// TwinCAT 3 PLC project PlcIotHttpSamplesPhilipsHue
// ProgramVersion: 3.1.4026.25
// libraries:
//   Tc2_Standard, * (Beckhoff Automation GmbH)
//   Tc2_System, * (Beckhoff Automation GmbH)
//   Tc2_Utilities, * (Beckhoff Automation GmbH)
//   Tc3_IotBase, * (Beckhoff Automation GmbH)
//   Tc3_JsonXml, * (Beckhoff Automation GmbH)
//   Tc3_Module, * (Beckhoff Automation GmbH)
// project tree:
//   / PlcTask.TcTTO (not stored)
//   POUs/ MAIN.TcPOU
//   POUs/Philips Hue/ FB_TestHTTP_Put_PhilipsHue.TcPOU
// real-time tasks:
//   TASK PlcTask: cycle T#10ms, priority 24, ADS port 350

// ---- POUs/MAIN.TcPOU
PROGRAM MAIN
VAR
	// trigger command execution for Philips Hue samples
	bPutPhilipsHue 					: BOOL;

	fbHttpClientPhilipsHue			: FB_IotHttpClient := (sHostName := '192.168.0.100',
									bKeepAlive := TRUE, tConnectionTimeout := T#10S);

	fbHttpPutPhilipsHue				: FB_TestHTTP_Put_PhilipsHue;
	
	bBlinkingMode					: BOOL;
	fbTimer							: TON:=(PT:=T#500MS);
	nColor               			: UINT;
END_VAR

// init client parameters at startup
IF NOT fbHttpClientPhilipsHue.bConfigured THEN 
	fbHttpClientPhilipsHue.nHostPort := 443;
	fbHttpClientPhilipsHue.stTLS.bNoServerCertCheck := TRUE;
END_IF

IF fbHttpClientPhilipsHue.bConfigured THEN
	fbHttpPutPhilipsHue(bSend := bPutPhilipsHue, fbClient := fbHttpClientPhilipsHue, nColor := nColor);
END_IF

IF bBlinkingMode THEN
	fbTimer(IN := NOT fbTimer.Q);
	IF fbTimer.Q THEN
		nColor := nColor +5000;
		IF nColor = 65000 THEN
			nColor :=0;
		END_IF
		IF bPutPhilipsHue THEN
			bPutPhilipsHue := FALSE;
		ELSE 
			bPutPhilipsHue := TRUE;
		END_IF
	END_IF
END_IF

fbHttpClientPhilipsHue.Execute();

END_PROGRAM

// ---- POUs/Philips Hue/FB_TestHTTP_Put_PhilipsHue.TcPOU
FUNCTION_BLOCK FB_TestHTTP_Put_PhilipsHue
VAR_INPUT
	bSend				: BOOL;
	nColor				: UINT;
END_VAR
VAR_IN_OUT
	fbClient			: FB_IotHttpClient;
END_VAR
VAR_OUTPUT
	bBusy				: BOOL;
	bError				: BOOL;
END_VAR
VAR
	fbRequest			: FB_IotHttpRequest;
	fbJson				: FB_JsonDomParser;
	fbJsonWriter		: FB_JsonSaxWriter;
	nState				: UDINT;
	RisingEdge			: R_TRIG;
	
	bGetContentResult	: BOOL;
	sContent			: STRING(511);
	sSend				: STRING(255);
	
	bGetJsonResult		: BOOL;
	jsonDoc				: SJsonValue;
	
	nReqCount			: UDINT;	
	nResCount			: UDINT;
	nValidResCount		: UDINT;
	nErrCount			: UDINT;
END_VAR

RisingEdge(CLK := bSend );

CASE nState OF
0:	
	IF RisingEdge.Q THEN 
		fbJsonWriter.StartObject();
		fbJsonWriter.AddKey('on');
		fbJsonWriter.AddBool(TRUE);
		fbJsonWriter.AddKey('sat');
		fbJsonWriter.AddUdint(50);
		fbJsonWriter.AddKey('bri');
		fbJsonWriter.AddUdint(100);
		fbJsonWriter.AddKey('hue');
		fbJsonWriter.AddUdint(nColor);
		fbJsonWriter.EndObject();
		// If object is longer than 256 byte, CopyDocument method must be used
		sSend := fbJsonWriter.GetDocument();
		fbJsonWriter.ResetDocument();
		IF fbRequest.SendRequest(sUri := '/api/censored/lights/1/state' , fbClient := fbClient, eRequestType := ETcIotHttpRequestType.HTTP_PUT, pContent := ADR(sSend), nContentSize := LEN2(ADR(sSend)), 0) THEN				
			nState := 1;
			nReqCount := nReqCount +1;
			bBusy := TRUE;
			bError := FALSE;
		END_IF					
	END_IF
1:
	IF NOT fbRequest.bBusy THEN
		bError := TRUE;
		IF NOT fbRequest.bError THEN				 
			bGetContentResult := fbRequest.GetContent(pContent := ADR(sContent), nContentSize := SIZEOF(sContent), bSetNullTermination := TRUE);
			IF fbRequest.nStatusCode >= 200 AND fbRequest.nStatusCode < 300 THEN
				bGetJsonResult := FALSE;
				jsonDoc := fbRequest.GetJsonDomContent(fbJson);
				IF jsonDoc <> 0 THEN
					; // do something with status response
					nValidResCount := nValidResCount+1;
					bError := FALSE;	
				END_IF							
				nResCount := nResCount+1;			
			END_IF
		END_IF
		nState := 0;
		bBusy := FALSE;
		IF bError THEN
			nErrCount := nErrCount +1;
		END_IF
	END_IF  	
END_CASE

END_FUNCTION_BLOCK
